// TIA Portal V19 export
DATA_BLOCK "PID_Loops_DB"   // DB30
VERSION : 0.0
// stored: AutoNumber false, InstanceOfName PID HMI Interface, InstanceOfType FB
"PID HMI Interface"
   // VAR_INPUT
   //    LoopSelection : Int;
   // END_VAR
   // VAR_OUTPUT
   //    RPM : Real := 0.0;
   // END_VAR
   // VAR_IN_OUT
   //    Hmi : Struct
   //       PV : Real;
   //       SP : Real;
   //       EngUnitsMin : Real;
   //       EngUnitsMax : Real;
   //       P : Real;
   //       I : Time;
   //       D : Time;
   //       Auto_Man : Struct
   //          Auto : Bool;
   //          Manual : Bool;
   //          UpdateParaRec : Bool;
   //       END_STRUCT;
   //       MV : Real;
   //       OP : Real;
   //    END_STRUCT;
   //    PC : "M0940_PIDInterface";
   //    LC : "M0940_PIDInterface";
   // END_VAR
   // VAR
   //    PID_Loop : CONT_C;
   //    RatioFactor : Real := 0.0;
   //    PV_0_100 : Real := 0.0;
   //    SP_0_100 : Real := 0.0;
   //    LoopSelMem : Int;
   //    FP : Bool;
   // END_VAR
BEGIN
END_DATA_BLOCK
